# EPICS substitutions: extendsApp/Db/user.substitutions
# Example substitutions file

file "db/dbExample1.db" {
    { user = "parallels" }
}

file db/dbExample2.db {
    pattern { user, no, scan }
        { "parallels", 1, "1 second" }
        { "parallels", 2, "2 second" }
        { "parallels", 3, "5 second" }
}
